(* CoDeSys 2.3.9.35 project: tb4F.pro *)
(* Author: Hemerson *)
(* Libraries: SysLibTargetVisu.lib 26.11.08 09:50:36, Standard.lib 26.11.08 09:46:20, Iecsfc.lib 26.11.08 09:46:14, DU35x.lib 7.7.11 15:59:53, SYSLIBCALLBACK.LIB 26.11.08 09:50:38 *)

(* PLC configuration (modules and I/O channels)
PLC Configuration [Root] node -1, in %IB0 out %QB0
  Communication [Comunica] node 0, in %IB0 out %QB0
    COM1 [COM1] node 0, in %IB0 out %QB0 {BaudRate = 115200; Paridade = No Parity; StopBits = 1 Stop Bit; Modem = Without RTS/CTS; Delay = 5}
      MToolIEC [Codesys] node 0, in %IB0 out %QB0
    COM2 [COM2] node 1, in %IB0 out %QB0 {BaudRate = 115200; Paridade = No Parity; StopBits = 1 Stop Bit; Modem = Without RTS/CTS; Delay = 5}
      Disable [Desabilitado485] node 0, in %IB0 out %QB0
  Bus [Barramento] node 1, in %IB0 out %QB0
    Inputs [Entradas] node 0, in %IB0 out %QB0
      Digital Inputs 0 [Entradas0] node 0, in %IW0 out %QB0
        I00 AT %IX0.0 [BitInput] I0.0
        I01 AT %IX0.1 [BitInput] I0.1
        I02 AT %IX0.2 [BitInput] I0.2
        I03 AT %IX0.3 [BitInput] I0.3
        I04 AT %IX0.4 [BitInput] I0.4
        I05 AT %IX0.5 [BitInput] I0.5
        I06 AT %IX0.6 [BitInput] I0.6
        I07 AT %IX0.7 [BitInput] I0.7
        I08 AT %IX0.8 [BitInput] I0.8
      Digital Inputs 1 [Entradas1] node 0, in %IW1 out %QB0
        I10 AT %IX1.0 [BitInput] I1.0
        I11 AT %IX1.1 [BitInput] I1.1
        I12 AT %IX1.2 [BitInput] I1.2
        I13 AT %IX1.3 [BitInput] I1.3
        I14 AT %IX1.4 [BitInput] I1.4
        I15 AT %IX1.5 [BitInput] I1.5
        I16 AT %IX1.6 [BitInput] I1.6
        I17 AT %IX1.7 [BitInput] I1.7
        I18 AT %IX1.8 [BitInput] I1.8
      Digital Inputs 2 [Entradas2] node 0, in %IW2 out %QB0
        I20 AT %IX2.0 [BitInput] I2.0
        I21 AT %IX2.1 [BitInput] I2.1
      Analog Inputs [EntradaAnalogica] node 0, in %IW4 out %QB0
        AI0 AT %IW4 [WordInput] AI0 {TipoAnalogica = Channel Disable; FiltroAnalogica = Filter 0 - AI=2ms  / AV=90ms; FundoEscala = 0}
        AI1 AT %IW5 [WordInput] AI1 {TipoAnalogica = Channel Disable; FiltroAnalogica = Filter 0 - AI=2ms  / AV=90ms; FundoEscala = 0}
        AI2 AT %IW6 [WordInput] AI2 {TipoAnalogica = Channel Disable; FiltroAnalogica = Filter 0 - AI=2ms  / AV=90ms; FundoEscala = 0}
        AI3 AT %IW7 [WordInput] AI3 {TipoAnalogica = Channel Disable; FiltroAnalogica = Filter 0 - AI=2ms  / AV=90ms; FundoEscala = 0}
      Fast Inputs [EntradasRapidas] node 1, in %IB16 out %QB0
        Block 0 [Bloco0] node 0, in %IB16 out %QB0
          Disable [DesabilitadoBloco0] node 0, in %IB16 out %QB0
        Block 1 [Bloco1] node 1, in %IB16 out %QB0
          Disable [DesabilitadoBloco1] node 0, in %IB16 out %QB0
        Configurable Input Block 0 [EntradaConfiBloco0] node 2, in %IB16 out %QB0
          Counter 0 [EntradaConfContador0] node 0, in %IB16 out %QB0 {EntradaConfiguravelContador = Disable}
        Configurable Input Block 1 [EntradaConfiBloco1] node 3, in %IB16 out %QB0
          Counter 2 [EntradaConfContador2] node 0, in %IB16 out %QB0 {EntradaConfiguravelContador = Disable}
    Outputs [Saidas] node 1, in %IB13 out %QB0
      Digital Outputs 0 [Saidas0] node 0, in %IW0 out %QW0
        Q00 AT %QX0.0 [BitOutput] Q0.0
        Q01 AT %QX0.1 [BitOutput] Q0.1
        Q02 AT %QX0.2 [BitOutput] Q0.2
        Q03 AT %QX0.3 [BitOutput] Q0.3
        Q04 AT %QX0.4 [BitOutput] Q0.4
        Q05 AT %QX0.5 [BitOutput] Q0.5
        Q06 AT %QX0.6 [BitOutput] Q0.6
        Q07 AT %QX0.7 [BitOutput] Q0.7
      Digital Outputs 1 [Saidas1] node 0, in %IW0 out %QW1
        Q10 AT %QX1.0 [BitOutput] Q1.0
        Q11 AT %QX1.1 [BitOutput] Q1.1
        Q12 AT %QX1.2 [BitOutput] Q1.2
        Q13 AT %QX1.3 [BitOutput] Q1.3
        Q14 AT %QX1.4 [BitOutput] Q1.4
        Q15 AT %QX1.5 [BitOutput] Q1.5
        Q16 AT %QX1.6 [BitOutput] Q1.6
        Q17 AT %QX1.7 [BitOutput] Q1.7
      Analog Outputs [SaidaAnalogica] node 0, in %IW0 out %QW3
        AO0 AT %QW3 [WordOutput] AO0 {TipoAnalogica = Channel Disable; FundoEscala = 0}
        AO1 AT %QW4 [WordOutput] AO1 {TipoAnalogica = Channel Disable; FundoEscala = 0}
      Fast Outputs [SaidasRapidas] node 1, in %IB0 out %QB10
        Fast Output 0 Disable [DesabilitadoF0] node 0, in %IB0 out %QB10
        Fast Output 1 Disable [DesabilitadoF1] node 1, in %IB0 out %QB10
      Counter Output [SaidasContador] node 2, in %IB0 out %QB10
        Block 0 Output Disable [DesabilitadoSaidaBloco0] node 0, in %IB0 out %QB10
        Block 1 Output Disable [DesabilitadoSaidaBloco1] node 1, in %IB0 out %QB10
  External Events [Eventos] node 2, in %IB13 out %QB6
    Timer Event [TimerEvent] node 0, in %IB13 out %QB6 {Intervalo = 10}
*)

(* Global variable list: Variáveis globais *)
VAR_GLOBAL
	D  AT %IX0.0: BOOL;
	A1 AT %IX0.1: BOOL;
	A2 AT %IX0.2: BOOL;
	A3 AT %IX0.3: BOOL;
	A4 AT %IX0.4: BOOL;
	A5 AT %IX0.5: BOOL;
	A6 AT %IX0.6: BOOL;
	Q1: BOOL;
	Q2: BOOL;
	Q3: BOOL;
	Q4: BOOL;
	Q5: BOOL;
	Q6: BOOL;
	M1 AT %QX1.0: BOOL;
	M2 AT %QX1.1: BOOL;
	M3 AT %QX1.2: BOOL;
	M4 AT %QX1.3: BOOL;
	M5 AT %QX1.4: BOOL;
	M6 AT %QX1.5: BOOL;
	TEMP1: TON;
	TEMP2: TON;
	TEMP3: TON;
	M: BOOL;
	TEMP: TON;
	RESET_CLOCK: BOOL;
	DELAY: TON;
	START_CLOCK: BOOL;
	CLOCK: BOOL;
	CONTADOR: CTU;
	Q: BOOL;
	CONTADOR1: CTU;
	CONTADOR2: CTU;
	CONTADOR3: CTU;
	CONTADOR4: CTU;
	CONTADOR5: CTU;
	CONTADOR6: CTU;
	TRIG1: R_TRIG;
	TRIG2: R_TRIG;
	TRIG3: R_TRIG;
	TRIG4: R_TRIG;
	TRIG5: R_TRIG;
	TRIG6: R_TRIG;
	TRIG_A1: R_TRIG;
	TRIG_A2: R_TRIG;
	TRIG_A3: R_TRIG;
	TRIG_A4: R_TRIG;
	TRIG_A5: R_TRIG;
	TRIG_A6: R_TRIG;
	AUX:INT;
	SC1: BOOL;
	SC2: BOOL;
	SC3: BOOL;
	SC4: BOOL;
	SC5: BOOL;
	SC6: BOOL;
	RESET1: BOOL;
	RESET2: BOOL;
	RESET3: BOOL;
	RESET4: BOOL;
	RESET5: BOOL;
	RESET6: BOOL;
	RESET_P:BOOL;
	START_CONT: BOOL;
	CONTADOR_P: CTU;
	TRI: R_TRIG;
	SC_P: BOOL;
	CV_P: INT;
	PM1: INT;
	PM2: INT;
	PM3: INT;
	PM4: INT;	(*  *)
	PM5: INT;
	PM6: INT;


	SC_S: BOOL;
	RESET_S: BOOL;
	CONTADOR_S: CTU;

	TRI_S: R_TRIG;
	TRI_P: R_TRIG;
	START_CONT_S: BOOL;
	ON_CONT: BOOL;
	CV_S: INT;
	TV1: BOOL;
	TV2: BOOL;
	TV3: BOOL;
	TV4: BOOL;
	TV5: BOOL;
	TV6: BOOL;
	AUX1: BOOL;
	AUX2: BOOL;
	AUX3: BOOL;
	AUX4: BOOL;
	AUX5: BOOL;
	AUX6: BOOL;
END_VAR

(* POU PLC_PRG, LD *)
PROGRAM PLC_PRG
VAR
	D  AT %IX0.0: BOOL;
	A1 AT %IX0.1: BOOL;
	A2 AT %IX0.2: BOOL;
	A3 AT %IX0.3: BOOL;
	A4 AT %IX0.4: BOOL;
	A5 AT %IX0.5: BOOL;
	A6 AT %IX0.6: BOOL;
	Q1: BOOL;
	Q2: BOOL;
	Q3: BOOL;
	Q4: BOOL;
	Q5: BOOL;
	Q6: BOOL;
	M1 AT %QX1.0: BOOL;
	M2 AT %QX1.1: BOOL;
	M3 AT %QX1.2: BOOL;
	M4 AT %QX1.3: BOOL;
	M5 AT %QX1.4: BOOL;
	M6 AT %QX1.5: BOOL;
	TEMP1: TON;
	TEMP2: TON;
	TEMP3: TON;
	M: BOOL;
	TEMP: TON;
	RESET_CLOCK: BOOL;
	DELAY: TON;
	START_CLOCK: BOOL;
	CLOCK: BOOL;
	CONTADOR: CTU;
	Q: BOOL;
	CONTADOR1: CTU;
	CONTADOR2: CTU;
	CONTADOR3: CTU;
	CONTADOR4: CTU;
	CONTADOR5: CTU;
	CONTADOR6: CTU;
	TRIG1: R_TRIG;
	TRIG2: R_TRIG;
	TRIG3: R_TRIG;
	TRIG4: R_TRIG;
	TRIG5: R_TRIG;
	TRIG6: R_TRIG;
	TRIG_A1: R_TRIG;
	TRIG_A2: R_TRIG;
	TRIG_A3: R_TRIG;
	TRIG_A4: R_TRIG;
	TRIG_A5: R_TRIG;
	TRIG_A6: R_TRIG;
	AUX:INT;
	SC1: BOOL;
	SC2: BOOL;
	SC3: BOOL;
	SC4: BOOL;
	SC5: BOOL;
	SC6: BOOL;
	RESET1: BOOL;
	RESET2: BOOL;
	RESET3: BOOL;
	RESET4: BOOL;
	RESET5: BOOL;
	RESET6: BOOL;
	RESET_P:BOOL;
	START_CONT: BOOL;
	CONTADOR_P: CTU;
	TRI: R_TRIG;
	SC_P: BOOL;
	CV_P: INT;
	PM1: INT := 0;
	PM2: INT := 0;
	PM3: INT := 0;
	PM4: INT := 0;(*  *)
	PM5: INT := 0;
	PM6: INT := 0;


	SC_S: BOOL;
	RESET_S: BOOL;
	CONTADOR_S: CTU;

	TRI_S: R_TRIG;
	TRI_P: R_TRIG;
	START_CONT_S: BOOL;
	ON_CONT: BOOL;
	CV_S: INT;
	TV1: TIME;
	TV2: TIME;
	TV3: TIME;
	TV4: TIME;
	TV5: TIME;
	TV6: TIME;
	AUX1: BOOL;
	AUX2: BOOL;
	AUX3: BOOL;
	AUX4: BOOL;
	AUX5: BOOL;
	AUX6: BOOL;
	DELAY1: TON;
	DELAY3: TON;
	DELAY4: TON;
	TEMP6: TON;
	TEMP5: TON;
	TEMP4: TON;
END_VAR
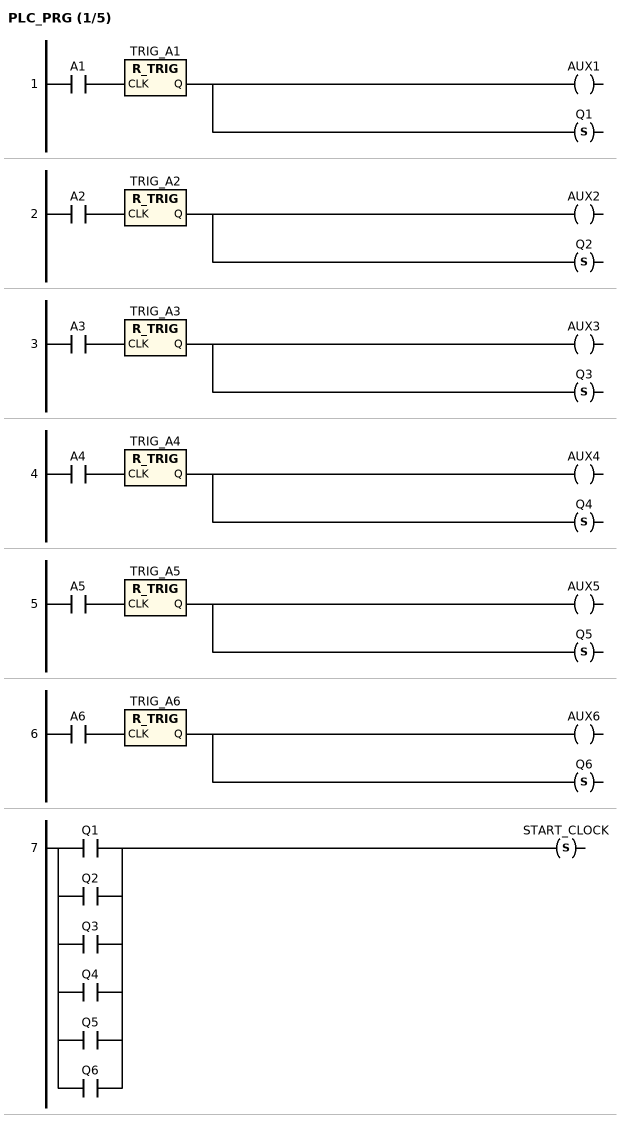
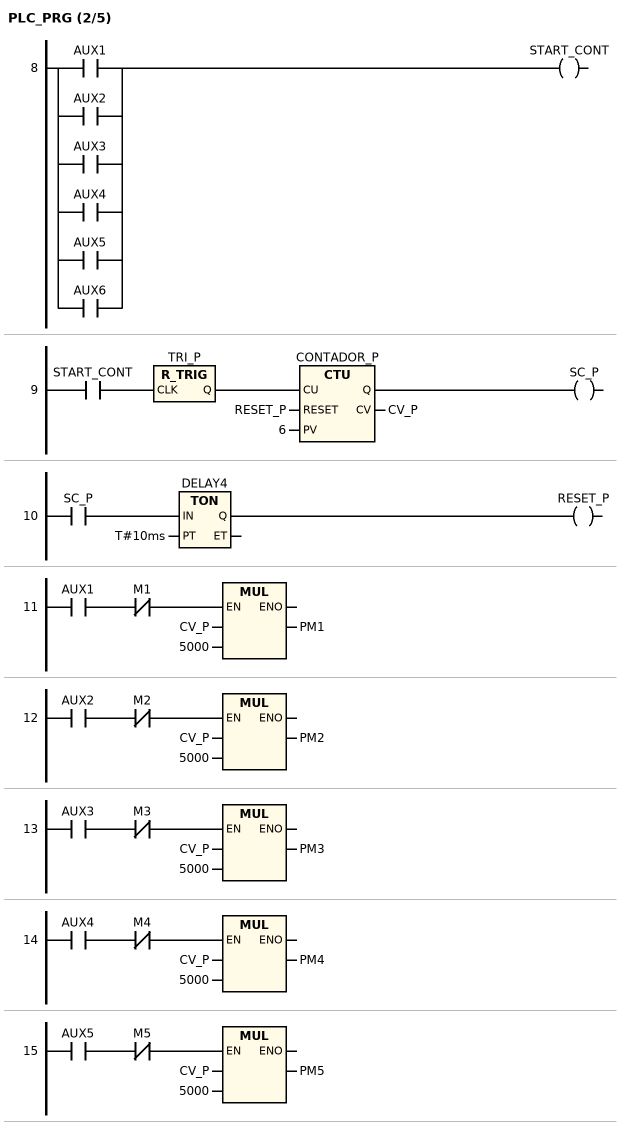
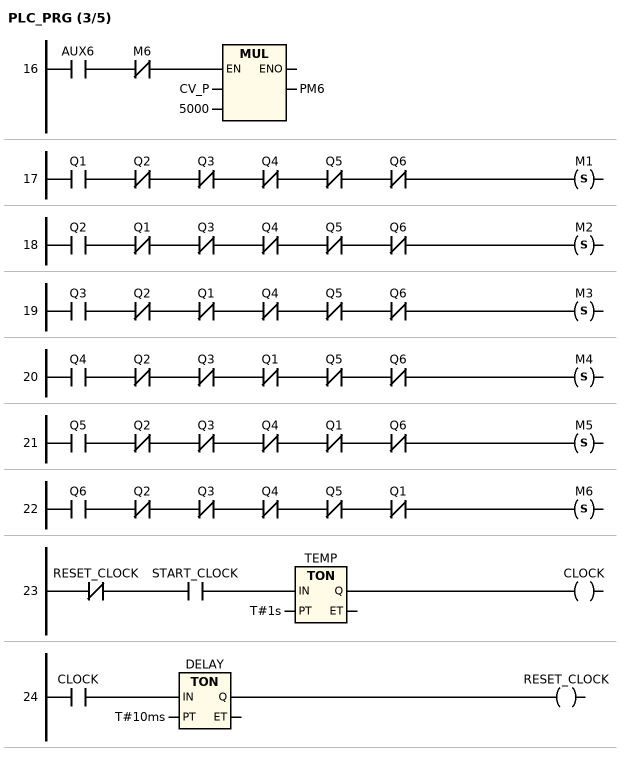
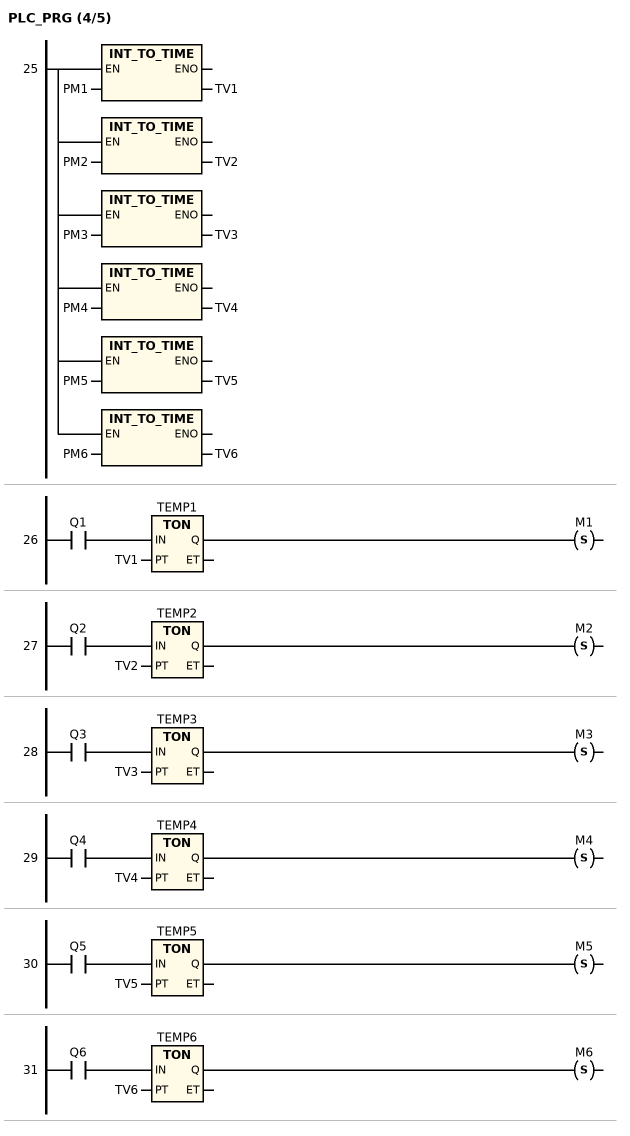
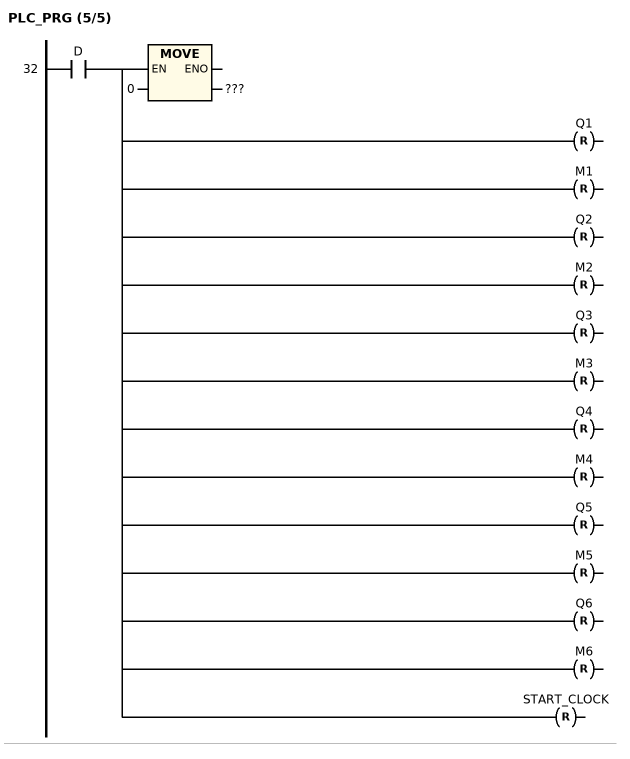
_LD_ (* Ladder Diagram *)
NETWORK 1
	[A1] - TRIG_A1:R_TRIG(CLK: *) --- (AUX1) (S Q1)
NETWORK 2
	[A2] - TRIG_A2:R_TRIG(CLK: *) --- (AUX2) (S Q2)
NETWORK 3
	[A3] - TRIG_A3:R_TRIG(CLK: *) --- (AUX3) (S Q3)
NETWORK 4
	[A4] - TRIG_A4:R_TRIG(CLK: *) --- (AUX4) (S Q4)
NETWORK 5
	[A5] - TRIG_A5:R_TRIG(CLK: *) --- (AUX5) (S Q5)
NETWORK 6
	[A6] - TRIG_A6:R_TRIG(CLK: *) --- (AUX6) (S Q6)
NETWORK 7
	{ [Q1] | [Q2] | [Q3] | [Q4] | [Q5] | [Q6] } --- (S START_CLOCK)
NETWORK 8
	{ [AUX1] | [AUX2] | [AUX3] | [AUX4] | [AUX5] | [AUX6] } --- (START_CONT)
NETWORK 9
	[START_CONT] - TRI_P:R_TRIG(CLK: *) - CONTADOR_P:CTU(CU: *, RESET: RESET_P, PV: 6, CV => CV_P) --- (SC_P)
NETWORK 10
	[SC_P] - DELAY4:TON(IN: *, PT: T#10ms) --- (RESET_P)
NETWORK 11
	[AUX1] - [/M1]
		EN --- MUL(CV_P, 5000) => PM1
NETWORK 12
	[AUX2] - [/M2]
		EN --- MUL(CV_P, 5000) => PM2
NETWORK 13
	[AUX3] - [/M3]
		EN --- MUL(CV_P, 5000) => PM3
NETWORK 14
	[AUX4] - [/M4]
		EN --- MUL(CV_P, 5000) => PM4
NETWORK 15
	[AUX5] - [/M5]
		EN --- MUL(CV_P, 5000) => PM5
NETWORK 16
	[AUX6] - [/M6]
		EN --- MUL(CV_P, 5000) => PM6
NETWORK 17
	[Q1] - [/Q2] - [/Q3] - [/Q4] - [/Q5] - [/Q6] --- (S M1)
NETWORK 18
	[Q2] - [/Q1] - [/Q3] - [/Q4] - [/Q5] - [/Q6] --- (S M2)
NETWORK 19
	[Q3] - [/Q2] - [/Q1] - [/Q4] - [/Q5] - [/Q6] --- (S M3)
NETWORK 20
	[Q4] - [/Q2] - [/Q3] - [/Q1] - [/Q5] - [/Q6] --- (S M4)
NETWORK 21
	[Q5] - [/Q2] - [/Q3] - [/Q4] - [/Q1] - [/Q6] --- (S M5)
NETWORK 22
	[Q6] - [/Q2] - [/Q3] - [/Q4] - [/Q5] - [/Q1] --- (S M6)
NETWORK 23
	[/RESET_CLOCK] - [START_CLOCK] - TEMP:TON(IN: *, PT: T#1s) --- (CLOCK)
NETWORK 24
	[CLOCK] - DELAY:TON(IN: *, PT: T#10ms) --- (RESET_CLOCK)
NETWORK 25
	*
		EN --- INT_TO_TIME(PM1) => TV1
		EN --- INT_TO_TIME(PM2) => TV2
		EN --- INT_TO_TIME(PM3) => TV3
		EN --- INT_TO_TIME(PM4) => TV4
		EN --- INT_TO_TIME(PM5) => TV5
		EN --- INT_TO_TIME(PM6) => TV6
NETWORK 26
	[Q1] - TEMP1:TON(IN: *, PT: TV1) --- (S M1)
NETWORK 27
	[Q2] - TEMP2:TON(IN: *, PT: TV2) --- (S M2)
NETWORK 28
	[Q3] - TEMP3:TON(IN: *, PT: TV3) --- (S M3)
NETWORK 29
	[Q4] - TEMP4:TON(IN: *, PT: TV4) --- (S M4)
NETWORK 30
	[Q5] - TEMP5:TON(IN: *, PT: TV5) --- (S M5)
NETWORK 31
	[Q6] - TEMP6:TON(IN: *, PT: TV6) --- (S M6)
NETWORK 32
	[D] --- (R Q1) (R M1) (R Q2) (R M2) (R Q3) (R M3) (R Q4) (R M4) (R Q5) (R M5) (R Q6) (R M6) (R START_CLOCK)
		EN --- MOVE(0) => ???
_END_LD_
(* the same logic as Structured Text *)
(* Network 1 *)
TRIG_A1(CLK := A1);
AUX1 := TRIG_A1.Q;
IF TRIG_A1.Q THEN Q1 := TRUE; END_IF;
(* Network 2 *)
TRIG_A2(CLK := A2);
AUX2 := TRIG_A2.Q;
IF TRIG_A2.Q THEN Q2 := TRUE; END_IF;
(* Network 3 *)
TRIG_A3(CLK := A3);
AUX3 := TRIG_A3.Q;
IF TRIG_A3.Q THEN Q3 := TRUE; END_IF;
(* Network 4 *)
TRIG_A4(CLK := A4);
AUX4 := TRIG_A4.Q;
IF TRIG_A4.Q THEN Q4 := TRUE; END_IF;
(* Network 5 *)
TRIG_A5(CLK := A5);
AUX5 := TRIG_A5.Q;
IF TRIG_A5.Q THEN Q5 := TRUE; END_IF;
(* Network 6 *)
TRIG_A6(CLK := A6);
AUX6 := TRIG_A6.Q;
IF TRIG_A6.Q THEN Q6 := TRUE; END_IF;
(* Network 7 *)
IF Q1 OR Q2 OR Q3 OR Q4 OR Q5 OR Q6 THEN START_CLOCK := TRUE; END_IF;
(* Network 8 *)
START_CONT := AUX1 OR AUX2 OR AUX3 OR AUX4 OR AUX5 OR AUX6;
(* Network 9 *)
TRI_P(CLK := START_CONT);
CONTADOR_P(CU := TRI_P.Q, RESET := RESET_P, PV := 6);
CV_P := CONTADOR_P.CV;
SC_P := CONTADOR_P.Q;
(* Network 10 *)
DELAY4(IN := SC_P, PT := T#10ms);
RESET_P := DELAY4.Q;
(* Network 11 *)
IF AUX1 AND NOT M1 THEN
	PM1 := CV_P * 5000;
END_IF;
(* Network 12 *)
IF AUX2 AND NOT M2 THEN
	PM2 := CV_P * 5000;
END_IF;
(* Network 13 *)
IF AUX3 AND NOT M3 THEN
	PM3 := CV_P * 5000;
END_IF;
(* Network 14 *)
IF AUX4 AND NOT M4 THEN
	PM4 := CV_P * 5000;
END_IF;
(* Network 15 *)
IF AUX5 AND NOT M5 THEN
	PM5 := CV_P * 5000;
END_IF;
(* Network 16 *)
IF AUX6 AND NOT M6 THEN
	PM6 := CV_P * 5000;
END_IF;
(* Network 17 *)
IF Q1 AND NOT Q2 AND NOT Q3 AND NOT Q4 AND NOT Q5 AND NOT Q6 THEN M1 := TRUE; END_IF;
(* Network 18 *)
IF Q2 AND NOT Q1 AND NOT Q3 AND NOT Q4 AND NOT Q5 AND NOT Q6 THEN M2 := TRUE; END_IF;
(* Network 19 *)
IF Q3 AND NOT Q2 AND NOT Q1 AND NOT Q4 AND NOT Q5 AND NOT Q6 THEN M3 := TRUE; END_IF;
(* Network 20 *)
IF Q4 AND NOT Q2 AND NOT Q3 AND NOT Q1 AND NOT Q5 AND NOT Q6 THEN M4 := TRUE; END_IF;
(* Network 21 *)
IF Q5 AND NOT Q2 AND NOT Q3 AND NOT Q4 AND NOT Q1 AND NOT Q6 THEN M5 := TRUE; END_IF;
(* Network 22 *)
IF Q6 AND NOT Q2 AND NOT Q3 AND NOT Q4 AND NOT Q5 AND NOT Q1 THEN M6 := TRUE; END_IF;
(* Network 23 *)
TEMP(IN := NOT RESET_CLOCK AND START_CLOCK, PT := T#1s);
CLOCK := TEMP.Q;
(* Network 24 *)
DELAY(IN := CLOCK, PT := T#10ms);
RESET_CLOCK := DELAY.Q;
(* Network 25 *)
TV1 := INT_TO_TIME(PM1);
TV2 := INT_TO_TIME(PM2);
TV3 := INT_TO_TIME(PM3);
TV4 := INT_TO_TIME(PM4);
TV5 := INT_TO_TIME(PM5);
TV6 := INT_TO_TIME(PM6);
(* Network 26 *)
TEMP1(IN := Q1, PT := TV1);
IF TEMP1.Q THEN M1 := TRUE; END_IF;
(* Network 27 *)
TEMP2(IN := Q2, PT := TV2);
IF TEMP2.Q THEN M2 := TRUE; END_IF;
(* Network 28 *)
TEMP3(IN := Q3, PT := TV3);
IF TEMP3.Q THEN M3 := TRUE; END_IF;
(* Network 29 *)
TEMP4(IN := Q4, PT := TV4);
IF TEMP4.Q THEN M4 := TRUE; END_IF;
(* Network 30 *)
TEMP5(IN := Q5, PT := TV5);
IF TEMP5.Q THEN M5 := TRUE; END_IF;
(* Network 31 *)
TEMP6(IN := Q6, PT := TV6);
IF TEMP6.Q THEN M6 := TRUE; END_IF;
(* Network 32: see the listing above *)
END_PROGRAM

(* Visualisation main
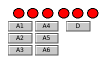
ellipse at (9,8)-(20,18): alarm colour if PLC_PRG.M1
ellipse at (23,8)-(34,18): alarm colour if PLC_PRG.M2
ellipse at (38,8)-(49,18): alarm colour if PLC_PRG.M3
button at (4,21)-(28,31): text "A1"; toggles PLC_PRG.A1
button at (4,33)-(28,43): text "A2"; toggles PLC_PRG.A2
button at (4,45)-(28,55): text "A3"; toggles PLC_PRG.A3
button at (31,21)-(54,31): text "A4"; toggles PLC_PRG.A4
button at (31,33)-(54,43): text "A5"; toggles PLC_PRG.A5
button at (31,45)-(54,55): text "A6"; toggles PLC_PRG.A6
button at (62,21)-(86,31): text "D"; toggles PLC_PRG.D
ellipse at (54,8)-(65,18): alarm colour if PLC_PRG.M4
ellipse at (68,8)-(79,18): alarm colour if PLC_PRG.M5
ellipse at (83,8)-(94,18): alarm colour if PLC_PRG.M6
*)
